(* NC axis ctrl for AX5000 via EtherCAT *)
FUNCTION_BLOCK FB_MC2_AX5000AxisCtrl
VAR_INPUT
	bEnable				: BOOL;		(* set TRUE to enable axis and drive *)
	bReset				: BOOL;		(* set TRUE to reset axis or drive from ERROR condition, min 100ms pulse length *)

	bEnableRevDir			: BOOL;		(* set TRUE to allow axis to run in reverse direction *)
	fOverride				: LREAL;	(* max axis output in % *)
	nEtherCATState		: UINT;		(* EtherCAT operating state *)
	(*bCalibrateAxis			: BOOL;*)
	(*bCalibrateSensorExist	: BOOL;*)

	bFastStop				: BOOL;		(* set TRUE to override RUN signals and stop axis immediately *)
	(*stAxisControl		: ST_AXIS_Control;*)

	eMotionType		: E_AXIS_MotionType;
	(*bRunAxis			: BOOL;	(*execute run*)*)
	fDistance			: LREAL;	(*target relative position*)
	fPosition			: LREAL;	(*target absolute position*)
	fSetVelo			: LREAL;	(* target velocity *)
	bStopAtPos		: BOOL;	(* set TRUE to stop at specified pos, set FALSE to stop immediately *)
	fStopPos			: LREAL;	(* target modulo stop position *)

	bJogFwd			: BOOL;		(* set TRUE to jog forwards *)
	bJogRev			: BOOL;		(* set TRUE to jog reverse *)
	fJogVelo			: LREAL;	(* jog velocity (does not take effect if jog is in progress *)

	(*stRamps				: ST_AxisCtrlRamps;	(* ramps for FastStop, Normal and Jog *)*)

	bSafetyNotOK			: BOOL;
	bCalibrateSyncImpulse	: BOOL;
END_VAR
VAR_IN_OUT
	stAxisConfig			: ST_AXIS_Config;
	stParamSet			: ST_AxisParameterSet;	(* NC axis parameter set *)
	stAxis				: AXIS_REF;	(* NC axis structure *)
END_VAR
VAR_OUTPUT
	bInitOK				: BOOL;		(* TRUE = parameter set read at least once *)
	bEnabled			: BOOL;		(* TRUE = axis is enabled *)
	bActive				: BOOL;		(* TRUE = axis is moving *)
	bHomeActive			: BOOL;
	bVeloActive			: BOOL;
	bAbsActive			: BOOL;
	bRelActive			: BOOL;
	bJogActive			: BOOL;		(* TRUE = axis is moving in JOG mode *)
	bRunningFwd			: BOOL;		(* TRUE = axis is running forwards *)
	bRunningRev			: BOOL;		(* TRUE = axis is running backwards *)
	bCalibrated			: BOOL;		(*TRUE = axis has benn calibrated*)
	(*bHomed				: BOOL;*)		(* TRUE = axis has been homed *)
	bAxisError			: BOOL;		(* TRUE = axis is in error state *)
	nAxisErrorID		: UDINT;	(* NC axis error code *)
	fActPos				: LREAL;	(* axis absolute position *)
	fModuloPos			: LREAL;	(* axis modulo position *)
	fActVelo			: LREAL;	(* axis act ual velocity *)
	bDriveError			: BOOL;		(* TRUE = drive is in error state *)
	nStatusDWord		: DWORD;	(* drive status code *)
	fDCLinkVolts		: LREAL;	(* DC link voltage (volts) *)
	fAmplifierTemp		: LREAL;	(* Amplifier temperature (degrees) *)
END_VAR
VAR
	(*bRunVelo			: BOOL;		(* set TRUE to run axis at specified velocity *)
	bRunAbsolute		: BOOL;		(* set TRUE to run axis at specified position *)
	bRunRelative		: BOOL;		(* set TRUE to run axis at specified distance *)*)

	bTest : BOOL;
	bAxisReset		: BOOL;
	bDriveReset		: BOOL;

	ftrigSaftyReset			: F_TRIG;
	fbAxisCtrl				: FB_MC2_BasicAxisCtrl;
	fbEtherCATDelay		: TON;
	fbAxisHome			: MC_Home;
	fbVeloCtrl				: FB_MC2_VeloCtrl;
	fbAbsCtrl				: FB_MC2_AbsCtrl;
	fbRelCtrl				: FB_MC2_RelCtrl;
	fbDriveReset			: FB_SoEReset;
	fbDriveStatus			: FB_MC2_AX5000Status;
END_VAR
(*
-------------------------------------------------------------------------------------------------
Date		Version	Author	Comments
-------------------------------------------------------------------------------------------------
30/01/2015	3.00.00	PB		Updated with new FB_MC2_BasicAxisCtrl
							FB_SoEReset for DriveReset now phased with fbSyncTimer in FB_MC2_BasicAxisCtrl
							FB_SoERead for strDriveStatus and nDriveStatusCode now phased with fbSyncTimer in FB_MC2_BasicAxisCtrl

-------------------------------------------------------------------------------------------------
18/05/2012	1.09.00	PB		FB_MC_AxisCtrl replaced by FB_MC2_BasicAxisCtrl and FB_MC2_VeloCtrl
17/01/2011	1.06.00	PB		5 cycle delay added between EtherCAT OP mode and bInitOK flag
23/09/2010	1.00.01	PB		Comms status added to bInitOK flag
05/02/2010	1.00.00	PB		Initial release

-------------------------------------------------------------------------------------------------
*)
VAR // added by the converter: edge detectors and wires of the graphical bodies
    _w1, _w2 : BOOL;
END_VAR

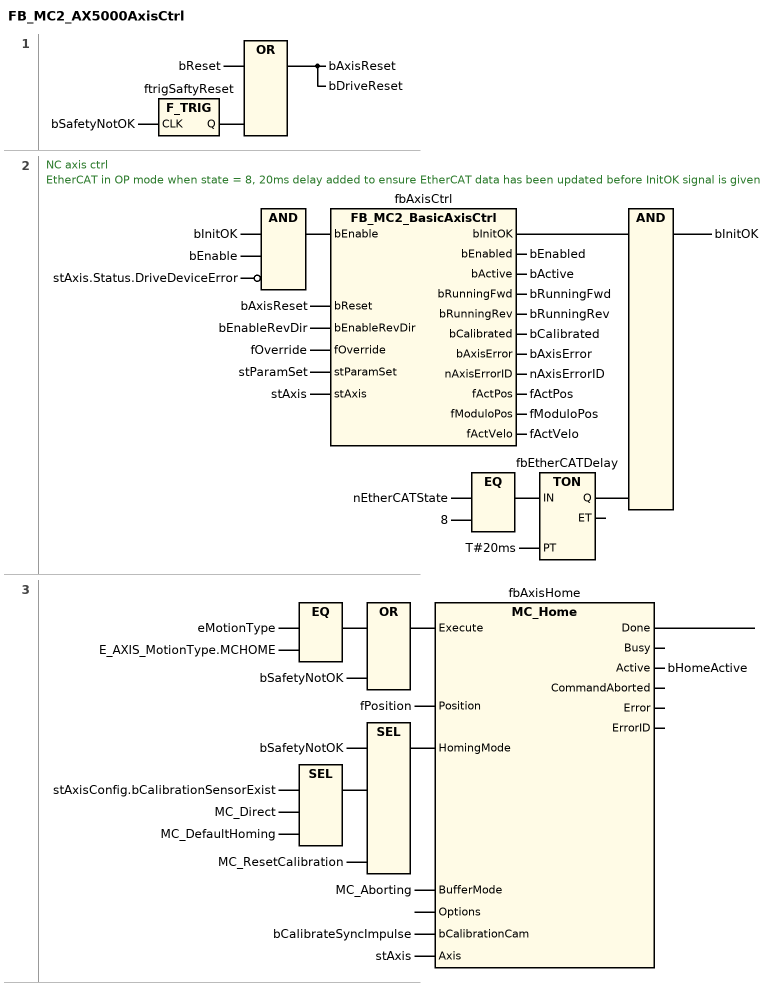
// NETWORK 1
ftrigSaftyReset(CLK := bSafetyNotOK); // F_TRIG
_w1 := bReset OR ftrigSaftyReset.Q;
bAxisReset := _w1;
bDriveReset := _w1;

// NETWORK 2
// 					NC axis ctrl
// EtherCAT in OP mode when state = 8, 20ms delay added to ensure EtherCAT data has been updated before InitOK signal is given
//
fbAxisCtrl(
    bEnable := bInitOK AND bEnable AND NOT stAxis.Status.DriveDeviceError,
    bReset := bAxisReset,
    bEnableRevDir := bEnableRevDir,
    fOverride := fOverride,
    stParamSet := stParamSet,
    stAxis := stAxis,
    bEnabled => bEnabled,
    bActive => bActive,
    bRunningFwd => bRunningFwd,
    bRunningRev => bRunningRev,
    bCalibrated => bCalibrated,
    bAxisError => bAxisError,
    nAxisErrorID => nAxisErrorID,
    fActPos => fActPos,
    fModuloPos => fModuloPos,
    fActVelo => fActVelo); // FB_MC2_BasicAxisCtrl
fbEtherCATDelay(IN := nEtherCATState = 8, PT := T#20ms); // TON
bInitOK := fbAxisCtrl.bInitOK AND fbEtherCATDelay.Q;

// NETWORK 3
fbAxisHome(
    Execute := eMotionType = E_AXIS_MotionType.MCHOME OR bSafetyNotOK,
    Position := fPosition,
    HomingMode := SEL(bSafetyNotOK, SEL(stAxisConfig.bCalibrationSensorExist, MC_Direct, MC_DefaultHoming), MC_ResetCalibration),
    BufferMode := MC_Aborting,
    bCalibrationCam := bCalibrateSyncImpulse,
    Axis := stAxis,
    Active => bHomeActive); // MC_Home

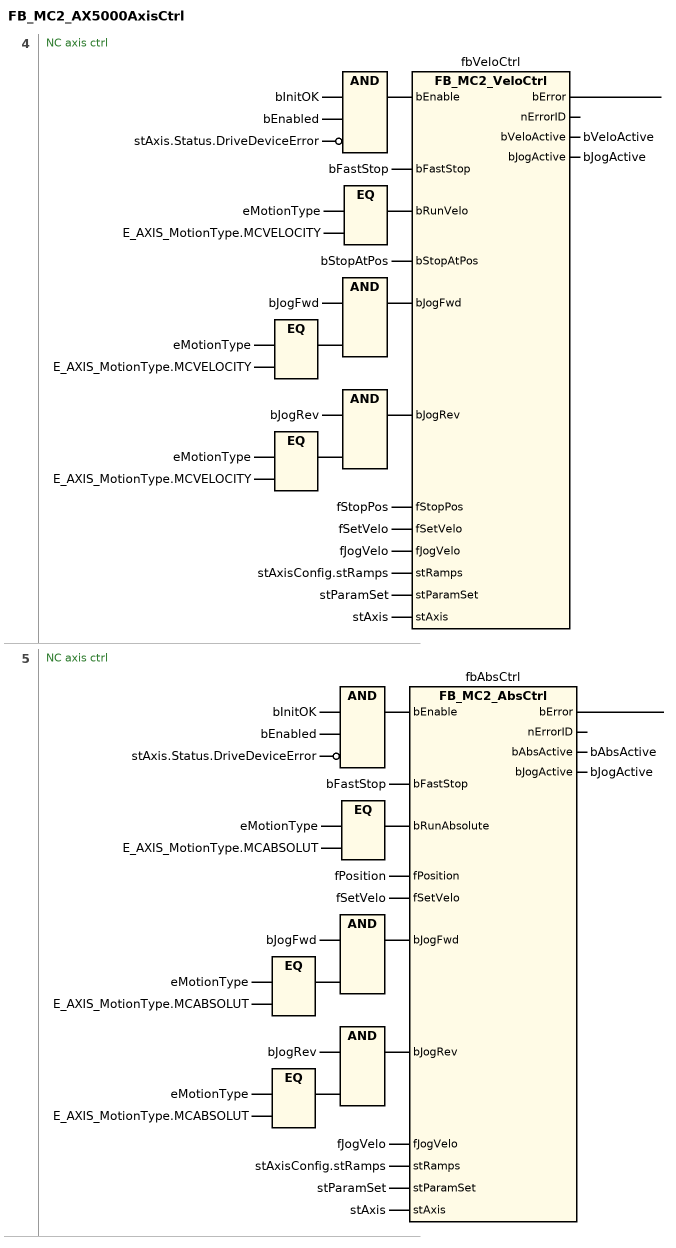
// NETWORK 4
// NC axis ctrl
fbVeloCtrl(
    bEnable := bInitOK AND bEnabled AND NOT stAxis.Status.DriveDeviceError,
    bFastStop := bFastStop,
    bRunVelo := eMotionType = E_AXIS_MotionType.MCVELOCITY,
    bStopAtPos := bStopAtPos,
    bJogFwd := bJogFwd AND eMotionType = E_AXIS_MotionType.MCVELOCITY,
    bJogRev := bJogRev AND eMotionType = E_AXIS_MotionType.MCVELOCITY,
    fStopPos := fStopPos,
    fSetVelo := fSetVelo,
    fJogVelo := fJogVelo,
    stRamps := stAxisConfig.stRamps,
    stParamSet := stParamSet,
    stAxis := stAxis,
    bVeloActive => bVeloActive,
    bJogActive => bJogActive); // FB_MC2_VeloCtrl

// NETWORK 5
// NC axis ctrl
fbAbsCtrl(
    bEnable := bInitOK AND bEnabled AND NOT stAxis.Status.DriveDeviceError,
    bFastStop := bFastStop,
    bRunAbsolute := eMotionType = E_AXIS_MotionType.MCABSOLUT,
    fPosition := fPosition,
    fSetVelo := fSetVelo,
    bJogFwd := bJogFwd AND eMotionType = E_AXIS_MotionType.MCABSOLUT,
    bJogRev := bJogRev AND eMotionType = E_AXIS_MotionType.MCABSOLUT,
    fJogVelo := fJogVelo,
    stRamps := stAxisConfig.stRamps,
    stParamSet := stParamSet,
    stAxis := stAxis,
    bAbsActive => bAbsActive,
    bJogActive => bJogActive); // FB_MC2_AbsCtrl

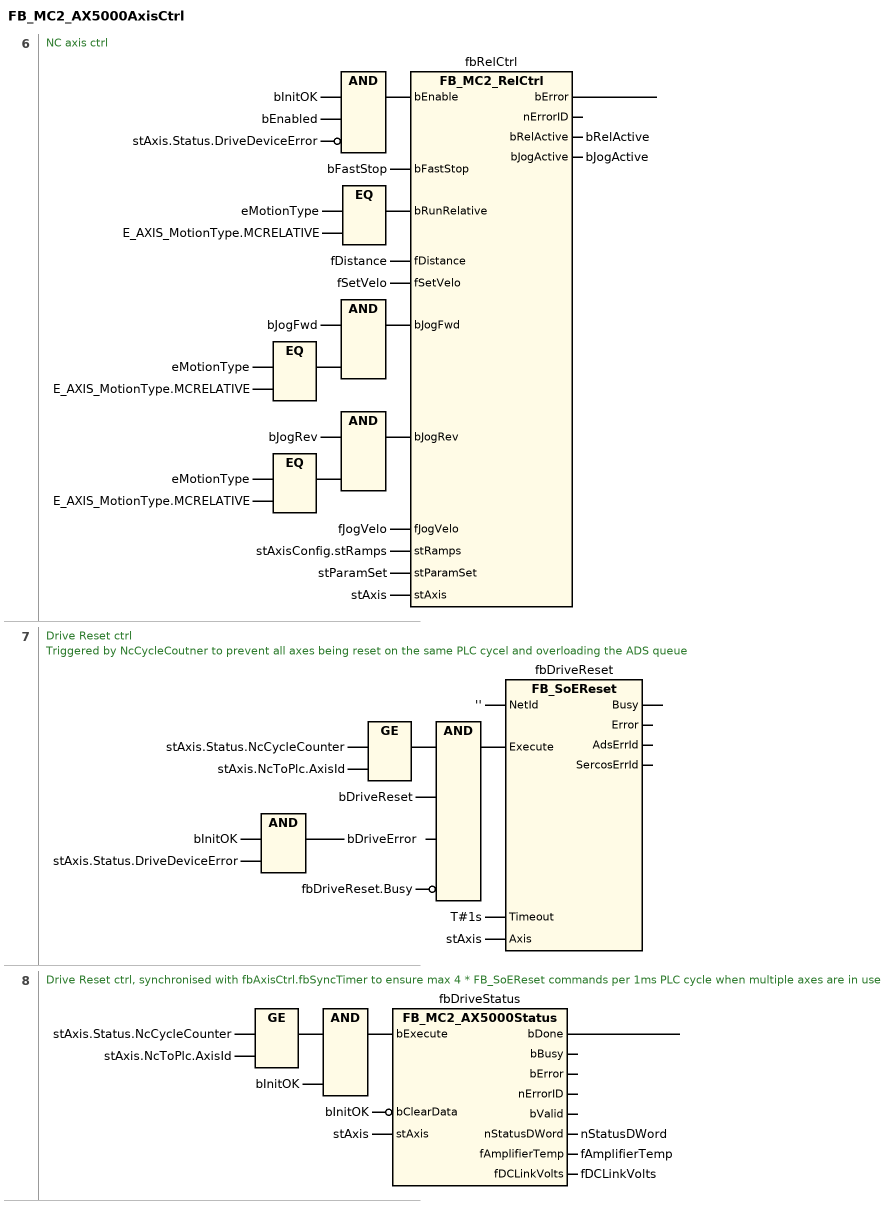
// NETWORK 6
// NC axis ctrl
fbRelCtrl(
    bEnable := bInitOK AND bEnabled AND NOT stAxis.Status.DriveDeviceError,
    bFastStop := bFastStop,
    bRunRelative := eMotionType = E_AXIS_MotionType.MCRELATIVE,
    fDistance := fDistance,
    fSetVelo := fSetVelo,
    bJogFwd := bJogFwd AND eMotionType = E_AXIS_MotionType.MCRELATIVE,
    bJogRev := bJogRev AND eMotionType = E_AXIS_MotionType.MCRELATIVE,
    fJogVelo := fJogVelo,
    stRamps := stAxisConfig.stRamps,
    stParamSet := stParamSet,
    stAxis := stAxis,
    bRelActive => bRelActive,
    bJogActive => bJogActive); // FB_MC2_RelCtrl

// NETWORK 7
// 					Drive Reset ctrl
// Triggered by NcCycleCoutner to prevent all axes being reset on the same PLC cycel and overloading the ADS queue
//
_w2 := bInitOK AND stAxis.Status.DriveDeviceError;
bDriveError := _w2;
fbDriveReset(
    NetId := '',
    Execute := stAxis.Status.NcCycleCounter >= stAxis.NcToPlc.AxisId AND bDriveReset AND _w2 AND NOT fbDriveReset.Busy,
    Timeout := T#1s,
    Axis := stAxis); // FB_SoEReset

// NETWORK 8
// Drive Reset ctrl, synchronised with fbAxisCtrl.fbSyncTimer to ensure max 4 * FB_SoEReset commands per 1ms PLC cycle when multiple axes are in use
fbDriveStatus(
    bExecute := stAxis.Status.NcCycleCounter >= stAxis.NcToPlc.AxisId AND bInitOK,
    bClearData := NOT bInitOK,
    stAxis := stAxis,
    nStatusDWord => nStatusDWord,
    fAmplifierTemp => fAmplifierTemp,
    fDCLinkVolts => fDCLinkVolts); // FB_MC2_AX5000Status

END_FUNCTION_BLOCK

(* stored: Version 1.1.0.1
   POU FB_MC2_AX5000AxisCtrl: Id {a2b20806-817a-404a-b050-32ae9941c146}, SpecialFunc None *)
